FUNCTION_BLOCK FB_A_Motor1R IMPLEMENTS I_Motor1R
VAR_INPUT
	I_iModus			:INT;		// Zustand des Systems (z.B. 0 = AUS | 1 = MAN | 2 = AUTO | 3 = Error)
	I_bVerriegeln		:BOOL;		// Verriegelte Elemente sind nicht ansteuerbar
	I_bReset			:BOOL;		// Zustand des Baustein wird zurückgesetzt 
	I_iGeschw			:INT;		// Angabe über Soll-Geschwindigkeit
END_VAR

VAR_OUTPUT
	O_bPower			:BOOL;		// Relais wird geschalten um FU mit Spannung zu versorgen
	O_iDrz				:INT;		// Ausgabe der Drehzahl für den Motor (Umrechnen von Spannung zu Drz)
	O_bStoerung			:BOOL;		// Befindet sich das Element in einem Error
	O_iStoerungID		:INT;		// Anzeigen von Störung über eine INT-Variable
END_VAR

VAR
	V_DrzMax		:INT;		// Variable für internes handling der Eigenschaft 
	V_Zeit			:TIME;		// Variable für internes handling der Eigenschaft 
	V_Status		:INT;		// Variable für internes handling der Eigenschaft 
	
	V_Timer			:TON;		// Runtime des Bausteins ermitteln
	
END_VAR

// Setzen der internen Variablen
P_MaxDrz := V_DrzMax;
V_Zeit := P_Laufzeit;
V_Status := P_Status;

// Reset des Bausteins
IF I_bReset THEN
	O_bStoerung := FALSE;
	O_iStoerungID := 0;
END_IF

// Verriegeln des Systems (Element geht in definierten Zustand) -> Motor wird gestoppt und ausgeschalten
IF I_bVerriegeln THEN
	O_iDrz := 0;
	O_bPower := FALSE;
END_IF

METHOD M_A_AN : BOOL
VAR_INPUT
END_VAR
// EBENE 1: Verriegelung
IF NOT I_bVerriegeln THEN	
	// EBEN 2: AUTO-Modus
		IF I_iModus = 2 THEN
			O_bPower := TRUE;
		END_IF
ELSE 
	O_bPower := FALSE;
END_IF

M_A_AN := O_bPower;
END_METHOD

METHOD M_A_AUS : BOOL
VAR_INPUT
END_VAR
IF I_iModus = 2 THEN
	O_bPower := FALSE;
	O_iDrz := 0;
END_IF

M_A_AUS := NOT O_bPower;
END_METHOD

METHOD M_A_START : BOOL
VAR_INPUT
END_VAR
// EBENE 1: Verriegelung
IF NOT I_bVerriegeln THEN

	// EBENE 2: Check der Drehzzahl
	IF I_iGeschw <= V_DrzMax THEN
		
		// Ebene 3: AUTO-Modus
		IF I_iModus = 2 THEN
			
			// EBENE 4: System muss AN sein
			IF O_bPower THEN
				O_iDrz := I_iGeschw;
				
			ELSE 	// Error: System ist nicht eingeschalten
				O_bStoerung := 1;
				O_iStoerungID := 11; 
		END_IF
		
	ELSE	// Error: Geschwindigkeit überschreitet die MaxDrz
		O_bStoerung := 1;
		O_iStoerungID := 12;
		END_IF		
	END_IF
END_IF

IF O_iDrz = I_iGeschw THEN
	M_A_START := TRUE;
ELSE
	M_A_START := FALSE;
END_IF
END_METHOD

METHOD M_A_STOP : BOOL
VAR_INPUT
END_VAR
// EBENE 1: Verriegelung
IF NOT I_bVerriegeln THEN
	O_iDrz := 0;
END_IF

IF O_iDrz = 0 THEN
	M_A_STOP := TRUE;
ELSE
	M_A_STOP := FALSE;
END_IF
END_METHOD

METHOD M_M_AN : BOOL
VAR_INPUT
END_VAR
// EBENE 1: Verriegelung
IF NOT I_bVerriegeln THEN	
	// EBEN 2: MAN-Modus
		IF I_iModus = 1 THEN
			O_bPower := TRUE;
		END_IF
ELSE 
	O_bPower := FALSE;
END_IF

M_M_AN := O_bPower;
END_METHOD

METHOD M_M_AUS : BOOL
VAR_INPUT
END_VAR
IF I_iModus = 1 THEN
	O_bPower := FALSE;
	O_iDrz := 0;
END_IF

M_M_AUS := NOT O_bPower;
END_METHOD

METHOD M_M_START : BOOL
VAR_INPUT
END_VAR
// EBENE 1: Verriegelung
IF NOT I_bVerriegeln THEN

	// EBENE 2: Check der Drehzzahl
	IF I_iGeschw <= V_DrzMax THEN
		
		// EBENE 3: MAN-Modus
		IF I_iModus = 1 THEN
			
			// EBENE 4: System muss AN sein
			IF O_bPower THEN
				O_iDrz := I_iGeschw;
				
			ELSE 	// Error: System ist nicht eingeschalten
				O_bStoerung := 1;
			O_iStoerungID := 11;
			END_IF
		END_IF
		
	ELSE	// Error: Geschwindigkeit überschreitet die MaxDrz
		O_bStoerung := 1;
		O_iStoerungID := 12;
	END_IF		
END_IF

IF O_iDrz = I_iGeschw THEN
	M_M_START := TRUE;
ELSE
	M_M_START := FALSE;
END_IF
END_METHOD

METHOD M_M_STOP : BOOL
VAR_INPUT
END_VAR
// EBENE 1: Verriegelung
IF NOT I_bVerriegeln THEN
	O_iDrz := 0;
END_IF

IF O_iDrz = 0 THEN
	M_M_STOP := TRUE;
ELSE
	M_M_STOP := FALSE;
END_IF
END_METHOD

PROPERTY PUBLIC P_Laufzeit : TIME
GET
IF O_iDrz > 0 THEN
	V_Timer(IN := TRUE, PT := T#100H);
END_IF

IF O_iDrz = 0 THEN
	V_Timer(IN := FALSE);
END_IF 
P_Laufzeit := V_Timer.ET;
END_GET
END_PROPERTY

PROPERTY PUBLIC P_MaxDrz : INT
SET
END_SET
END_PROPERTY

PROPERTY PUBLIC P_Status : INT
GET
IF O_bPower THEN
	P_Status := 1;
ELSE
	P_Status := 0;
END_IF

IF O_iDrz > 0 AND O_bPower THEN
	P_Status := 2;
ELSE
	P_Status := 1;
END_IF
END_GET
END_PROPERTY

END_FUNCTION_BLOCK

(* stored: Version 1.1.0.1, ProductVersion 3.1.4024.12
   POU FB_A_Motor1R: Id {512ae86b-4839-472c-9a02-ff7b77565c74}, SpecialFunc None
   Method M_A_AN: Id {65d9d92f-aa63-40be-bff0-334b4338033d}
   Method M_A_AUS: Id {5bcc46c0-7b79-45e9-aab7-8acecf003f61}
   Method M_A_START: Id {f235fccb-5b3c-4b37-992e-1ddc9f0cc742}
   Method M_A_STOP: Id {8268dcff-d4e4-49fd-9c65-0ffd9462f360}
   Method M_M_AN: Id {e2506041-3be8-4d33-9be8-63478ae299d0}
   Method M_M_AUS: Id {3a2bc3a2-7751-470f-9d31-99e6db741108}
   Method M_M_START: Id {6154265a-4a22-4203-8f36-ac3f14eef4f5}
   Method M_M_STOP: Id {7bf83711-66ca-4408-ae0d-b26a767e3151}
   Property P_Laufzeit: Id {18397b23-ad69-4f74-a52b-38ad0bf078f1}
   Get Get: Id {3ce4aceb-895c-4c68-991b-18a3443d2eff}
   Property P_MaxDrz: Id {86616c74-cb82-4b86-9dae-3431b2fbcd36}
   Set Set: Id {2f43768a-53ad-462b-9248-85b5781f7b51}
   Property P_Status: Id {4808de55-3ea3-4091-86d0-ecc11bc4a83b}
   Get Get: Id {cf1c6d07-f50d-408a-870d-7ab9c2dfa186} *)
